// TIA Portal V20 export
TYPE "typeEm3Standard"
// stored: Access Published, Namespace Unit1
   STRUCT
      commands { ExternalWritable := 'False'} : "Unit1.typeEm3Commands";
      monitoring { ExternalWritable := 'False'} : "Unit1.typeEm3Monitoring";
   END_STRUCT;
END_TYPE
